INTERFACE I_DefaultHomingBuilder EXTENDS __System.IQueryInterface

METHOD BuildDefaultHomingCommand : HomingCommand
END_METHOD

METHOD Cam : I_DefaultHomingBuilder
VAR_INPUT
	value : REFERENCE TO BOOL;
END_VAR
END_METHOD

METHOD ClearLag : I_PositioningHomingBuilder
END_METHOD

METHOD KeepLag : I_PositioningHomingBuilder
END_METHOD

METHOD Position : I_PositioningHomingBuilder
VAR_INPUT
	value : LREAL;
END_VAR
END_METHOD

METHOD ReferenceMode : I_DefaultHomingBuilder
VAR_INPUT
	value : EncoderReferenceMode;
END_VAR
END_METHOD

METHOD SearchDirection : I_DefaultHomingBuilder
VAR_INPUT
	value : Direction;
END_VAR
END_METHOD

METHOD SearchVelocity : I_DefaultHomingBuilder
VAR_INPUT
	value : LREAL;
END_VAR
END_METHOD

METHOD SyncDirection : I_DefaultHomingBuilder
VAR_INPUT
	value : Direction;
END_VAR
END_METHOD

METHOD SyncVelocity : I_DefaultHomingBuilder
VAR_INPUT
	value : LREAL;
END_VAR
END_METHOD

END_INTERFACE

(* stored: Version 1.1.0.1, ProductVersion 3.1.4026.13
   Itf I_DefaultHomingBuilder: Id {ba9c7290-0b01-0546-37b1-bdcfc7ebfe5f}
   Method BuildDefaultHomingCommand: Id {f6fe273c-6b44-0fd6-36f5-c85b3bb993ed}
   Method Cam: Id {d6036518-ee6b-0e7b-3972-9a49ecba1839}
   Method ClearLag: Id {f06544a2-96f3-0c9a-040f-8d5694e84d53}
   Method KeepLag: Id {0d23cecd-2b7e-08da-211e-0445fdcb987d}
   Method Position: Id {2c3e345e-4e45-0331-2788-8426551970b7}
   Method ReferenceMode: Id {97518c03-f4a6-0108-3526-6bcb62b73efd}
   Method SearchDirection: Id {2a8a16a7-6089-0c30-34a0-2bc82a81d0b2}
   Method SearchVelocity: Id {056f6655-6a83-0751-30e4-74d09a945a41}
   Method SyncDirection: Id {9a125247-e41a-0b24-2f99-2bb54a8a0b66}
   Method SyncVelocity: Id {78ad61b8-9d1d-012c-3fa8-58ee3fa6cd5d} *)
